Staubli VAL3: selectType.pgx

program selectType()
  local string l_sMessage
  local num l_nIndex
  local string l_sEvent
  local num l_nDefault
  local num l_nKey
  local num i
begin
  // change the processList
  call use:clear(0,13)
  call language:message(l_sMessage,191)
  call use:typeCenter(13,l_sMessage,40,true)
  call use:setSizeList(10,2,15,6)
  // build the list
  call use:listcreate(sMenu[4])
  call use:listadd(sType)
  call processList:getDefaultType(l_nDefault)
  call use:selectNewField(l_nDefault,0,0)
  // select the Item
  do
    l_nKey=get()
    call use:listevent(l_nKey,l_nIndex,l_sEvent)
  until l_nKey==270 or l_nKey==255
  if l_nKey==270
    call processList:setDefaultType(l_nIndex)
    use:bUseRefresh=true
  endIf
  //
end
